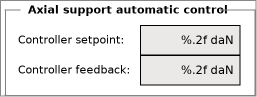
VISUALIZATION VISU_M1AxialSupportController  // 257x97
VAR_IN_OUT
	ref : M1AxialSupport;
    widget : M1AxialSupportWidget;
END_VAR
    Label (15,25 185x30), "Controller setpoint:"
    Label (15,55 185x30), "Controller feedback:"
    Rectangle (140,25 100x30), "%.2f daN", text variable: ref.controllerSetpoint.decaNewton.value
    Label (25,0 190x20), "Axial support automatic control"
    Rectangle (140,55 100x30), "%.2f daN", text variable: ref.mirrorAverageForce.average.decaNewton.value
    Polyline (20,10) (5,10) (5,95) (255,95) (255,10) (220,10)
END_VISUALIZATION

(* stored: Version 1.1.0.1, ProductVersion 3.1.4018.2
   Visu VISU_M1AxialSupportController: Id {b2eced71-c51b-4f93-9191-472a7b5602fe} *)
